// Interface for setting/ clearing local severity level.
INTERFACE I_EventSeverityHandler

// Clear the currently set local severity level.
METHOD ClearLocalSeverity
END_METHOD

// Get global severity level.
METHOD GetGlobalSeverity : TcEventSeverity
END_METHOD

// Get local severity level.
METHOD GetLocalSeverity : TcEventSeverity
END_METHOD

// Set a global severity level to filter logged events.
METHOD SetGlobalSeverity
VAR_INPUT
  severity : TcEventSeverity;
END_VAR
END_METHOD

// Set a local severity level to filter logged events. Ensure clear is called once local logging is complete.
METHOD SetLocalSeverity
VAR_INPUT
  severity : TcEventSeverity;
END_VAR
END_METHOD

END_INTERFACE

(* stored: Version 1.1.0.1, ProductVersion 3.1.4024.12
   Itf I_EventSeverityHandler: Id {2a5ac395-09d5-009d-1970-f6182d1fd6b4}
   Method ClearLocalSeverity: Id {469081a8-e859-0522-0475-5541fbbcfc5f}
   Method GetGlobalSeverity: Id {52d78de0-e695-0ab0-1818-1471bb8e09d7}
   Method GetLocalSeverity: Id {b245de1a-e2d1-09ac-16ea-cd645d5f528d}
   Method SetGlobalSeverity: Id {7d6a1756-8738-0df4-2144-4a14baa900c7}
   Method SetLocalSeverity: Id {8308f0e0-acda-0ad2-3df3-6b341102a394} *)
